SUBAPPLICATION Uebung_HystereseVertikal_AX_withAnalog (* MID/DEAD/HYSTERESIS-Eingabefelder bewegen live die 5 Schwellwert-Dreiecke im vertikalen Bargraph (Type=1 BottomToTop, Pixelposition gespiegelt: hoher Wert = kleiner Top) *)
  (* Standard: 61499-2; Description: Copyright (c) 2026 Meisterschulen am Ostbahnhof This program and the accompanying materials are made available under the terms of the Eclipse Public License 2.0 which is available at https://www.eclipse.org/legal/epl-2.0/ SPDX-License-Identifier: EPL-2.0 *)
  (* Version 1.1, 2026-09-27, Franz Höpfinger, Meisterschulen am Ostbahnhof, AR_TO_AI, Zero, QPos zu MyLib::sys::Q_ChildPosition_AR_Vertikal SubApp ausgelagert *)
  PACKAGE Uebungen;
  IMPORT Uebungen::const::UT::HystereseVertikal::DefaultPool_Numeric::InputNumber_MID_N;
  IMPORT Uebungen::const::UT::HystereseVertikal::DefaultPool_Numeric::InputNumber_DEAD_N;
  IMPORT Uebungen::const::UT::HystereseVertikal::DefaultPool_Numeric::InputNumber_HYSTERESIS_N;
  IMPORT Uebungen::const::UT::HystereseVertikal::DefaultPool::Polygon_MID;
  IMPORT Uebungen::const::UT::HystereseVertikal::DefaultPool::Polygon_MID_PLUS_DEAD;
  IMPORT Uebungen::const::UT::HystereseVertikal::DefaultPool::Polygon_MID_MINUS_DEAD;
  IMPORT Uebungen::const::UT::HystereseVertikal::DefaultPool::Polygon_MID_PLUS_DEAD_HYST;
  IMPORT Uebungen::const::UT::HystereseVertikal::DefaultPool::Polygon_MID_MINUS_DEAD_HYST;
  IMPORT Uebungen::const::UT::HystereseVertikal::DefaultPool::Container_Schwellwerte;
  IMPORT Uebungen::const::UT::HystereseVertikal::DefaultPool::NumberVariable_Istwert;
  IMPORT Uebungen::const::UT::HystereseVertikal::DefaultPool_Bargraph::Bargraph_Hysterese_ScalePx;
  IMPORT Uebungen::const::UT::HystereseVertikal::DefaultPool_Bargraph::Bargraph_Hysterese_LengthPx;
  IMPORT logiBUS::io::AI::logiBUS_AI::AnalogInput_I4;
  IMPORT logiBUS::io::DQ::logiBUS_DO::Output_Q1;
  IMPORT logiBUS::io::DQ::logiBUS_DO::Output_Q2;
  FBS
    MID_N : isobus::UT::io::NumericValue::NumericValue_PHYSA(QI := TRUE, stObj := InputNumber_MID_N);
    DEAD_N : isobus::UT::io::NumericValue::NumericValue_PHYSA(QI := TRUE, stObj := InputNumber_DEAD_N);
    HYST_N : isobus::UT::io::NumericValue::NumericValue_PHYSA(QI := TRUE, stObj := InputNumber_HYSTERESIS_N);
    Split_MID : adapter::events::unidirectional::AR_SPLIT_4;
    Split_DEAD : adapter::events::unidirectional::AR_SPLIT_3;
    Split_HYST : adapter::events::unidirectional::AR_SPLIT_3;
    Add_MidDead : adapter::iec61131::arithmetic::AR_ADD_2;
    Sub_MidDead : adapter::iec61131::arithmetic::AR_SUB_2;
    Split_AddResult : adapter::events::unidirectional::AR_SPLIT_2;
    Split_SubResult : adapter::events::unidirectional::AR_SPLIT_2;
    Add_MidDeadHyst : adapter::iec61131::arithmetic::AR_ADD_2;
    Sub_MidDeadHyst : adapter::iec61131::arithmetic::AR_SUB_2;
    AnalogInput_I4 : logiBUS::io::AI::logiBUS_AI_IDA(QI := TRUE, Input := AnalogInput_I4, AnalogInput_hysteresis := DWORD#0, TimeDelta := DWORD#250, TimeRateLimit := DWORD#100);
    AD_TO_AUDI : adapter::conversion::unidirectional::AD_TO_AUDI;
    AUDI_TO_AR : adapter::conversion::unidirectional::AUDI_TO_AR;
    Split_Istwert : adapter::events::unidirectional::AR_SPLIT_2;
    Q_Istwert : isobus::UT::Q::Q_NumericValue_PHYSA(stObj := (u16ObjId := NumberVariable_Istwert, r32Scale := 1.0, i32Offset := 0, u8Decimals := 0));
    DualHysteresis : logiBUS::signalprocessing::hysteresis::DualHysteresis_AR_AX(QI := TRUE);
    Output_Hoch : logiBUS::io::DQ::logiBUS_QXA(QI := TRUE, Output := Output_Q1);
    Output_Runter : logiBUS::io::DQ::logiBUS_QXA(QI := TRUE, Output := Output_Q2);
    BgLen_MID : adapter::types::unidirectional::AR::initval::initval_AR(INIT_VAL := Bargraph_Hysterese_LengthPx);
    SubFlip_MID : adapter::iec61131::arithmetic::AR_SUB_2;
    BgLen_MID_PLUS_DEAD : adapter::types::unidirectional::AR::initval::initval_AR(INIT_VAL := Bargraph_Hysterese_LengthPx);
    SubFlip_MID_PLUS_DEAD : adapter::iec61131::arithmetic::AR_SUB_2;
    BgLen_MID_MINUS_DEAD : adapter::types::unidirectional::AR::initval::initval_AR(INIT_VAL := Bargraph_Hysterese_LengthPx);
    SubFlip_MID_MINUS_DEAD : adapter::iec61131::arithmetic::AR_SUB_2;
    BgLen_MID_PLUS_DEAD_HYST : adapter::types::unidirectional::AR::initval::initval_AR(INIT_VAL := Bargraph_Hysterese_LengthPx);
    SubFlip_MID_PLUS_DEAD_HYST : adapter::iec61131::arithmetic::AR_SUB_2;
    BgLen_MID_MINUS_DEAD_HYST : adapter::types::unidirectional::AR::initval::initval_AR(INIT_VAL := Bargraph_Hysterese_LengthPx);
    SubFlip_MID_MINUS_DEAD_HYST : adapter::iec61131::arithmetic::AR_SUB_2;
  END_FBS
  SUBAPPS
    Mul_Istwert : MyLib::sys::AR_R_MUL(FACTOR := REAL#0.024420024420024420);
    Mul_MID : MyLib::sys::AR_R_MUL(FACTOR := Bargraph_Hysterese_ScalePx);
    QPos_MID : MyLib::sys::Q_ChildPosition_AR_Vertikal(u16ObjId := Polygon_MID, u16ObjIdParent := Container_Schwellwerte, xScale := TRUE);
    Mul_MID_PLUS_DEAD : MyLib::sys::AR_R_MUL(FACTOR := Bargraph_Hysterese_ScalePx);
    QPos_MID_PLUS_DEAD : MyLib::sys::Q_ChildPosition_AR_Vertikal(u16ObjId := Polygon_MID_PLUS_DEAD, u16ObjIdParent := Container_Schwellwerte, xScale := TRUE);
    Mul_MID_MINUS_DEAD : MyLib::sys::AR_R_MUL(FACTOR := Bargraph_Hysterese_ScalePx);
    QPos_MID_MINUS_DEAD : MyLib::sys::Q_ChildPosition_AR_Vertikal(u16ObjId := Polygon_MID_MINUS_DEAD, u16ObjIdParent := Container_Schwellwerte, xScale := TRUE);
    Mul_MID_PLUS_DEAD_HYST : MyLib::sys::AR_R_MUL(FACTOR := Bargraph_Hysterese_ScalePx);
    QPos_MID_PLUS_DEAD_HYST : MyLib::sys::Q_ChildPosition_AR_Vertikal(u16ObjId := Polygon_MID_PLUS_DEAD_HYST, u16ObjIdParent := Container_Schwellwerte, xScale := TRUE);
    Mul_MID_MINUS_DEAD_HYST : MyLib::sys::AR_R_MUL(FACTOR := Bargraph_Hysterese_ScalePx);
    QPos_MID_MINUS_DEAD_HYST : MyLib::sys::Q_ChildPosition_AR_Vertikal(u16ObjId := Polygon_MID_MINUS_DEAD_HYST, u16ObjIdParent := Container_Schwellwerte, xScale := TRUE);
  END_SUBAPPS
  ADAPTER_CONNECTIONS
    MID_N.rPhys TO Split_MID.IN;
    DEAD_N.rPhys TO Split_DEAD.IN;
    HYST_N.rPhys TO Split_HYST.IN;
    Split_MID.OUT2 TO Add_MidDead.IN1;
    Split_DEAD.OUT1 TO Add_MidDead.IN2;
    Split_MID.OUT3 TO Sub_MidDead.IN1;
    Split_DEAD.OUT2 TO Sub_MidDead.IN2;
    Add_MidDead.OUT TO Split_AddResult.IN;
    Sub_MidDead.OUT TO Split_SubResult.IN;
    Split_AddResult.OUT2 TO Add_MidDeadHyst.IN1;
    Split_HYST.OUT1 TO Add_MidDeadHyst.IN2;
    Split_SubResult.OUT2 TO Sub_MidDeadHyst.IN1;
    Split_HYST.OUT2 TO Sub_MidDeadHyst.IN2;
    AnalogInput_I4.IN TO AD_TO_AUDI.AD_IN;
    AD_TO_AUDI.AUDI_OUT TO AUDI_TO_AR.AUDI_IN;
    AUDI_TO_AR.AR_OUT TO Mul_Istwert.IN1;
    Mul_Istwert.OUT TO Split_Istwert.IN;
    Split_Istwert.OUT1 TO Q_Istwert.rPhys;
    Split_Istwert.OUT2 TO DualHysteresis.INPUT;
    Split_MID.OUT4 TO DualHysteresis.MI;
    Split_DEAD.OUT3 TO DualHysteresis.DEAD;
    Split_HYST.OUT3 TO DualHysteresis.HYSTERESIS;
    DualHysteresis.DO_UP TO Output_Hoch.OUT;
    DualHysteresis.DO_DOWN TO Output_Runter.OUT;
    Split_MID.OUT1 TO Mul_MID.IN1;
    BgLen_MID.OUT TO SubFlip_MID.IN1;
    Mul_MID.OUT TO SubFlip_MID.IN2;
    SubFlip_MID.OUT TO QPos_MID.rPhys;
    Split_AddResult.OUT1 TO Mul_MID_PLUS_DEAD.IN1;
    BgLen_MID_PLUS_DEAD.OUT TO SubFlip_MID_PLUS_DEAD.IN1;
    Mul_MID_PLUS_DEAD.OUT TO SubFlip_MID_PLUS_DEAD.IN2;
    SubFlip_MID_PLUS_DEAD.OUT TO QPos_MID_PLUS_DEAD.rPhys;
    Split_SubResult.OUT1 TO Mul_MID_MINUS_DEAD.IN1;
    BgLen_MID_MINUS_DEAD.OUT TO SubFlip_MID_MINUS_DEAD.IN1;
    Mul_MID_MINUS_DEAD.OUT TO SubFlip_MID_MINUS_DEAD.IN2;
    SubFlip_MID_MINUS_DEAD.OUT TO QPos_MID_MINUS_DEAD.rPhys;
    Add_MidDeadHyst.OUT TO Mul_MID_PLUS_DEAD_HYST.IN1;
    BgLen_MID_PLUS_DEAD_HYST.OUT TO SubFlip_MID_PLUS_DEAD_HYST.IN1;
    Mul_MID_PLUS_DEAD_HYST.OUT TO SubFlip_MID_PLUS_DEAD_HYST.IN2;
    SubFlip_MID_PLUS_DEAD_HYST.OUT TO QPos_MID_PLUS_DEAD_HYST.rPhys;
    Sub_MidDeadHyst.OUT TO Mul_MID_MINUS_DEAD_HYST.IN1;
    BgLen_MID_MINUS_DEAD_HYST.OUT TO SubFlip_MID_MINUS_DEAD_HYST.IN1;
    Mul_MID_MINUS_DEAD_HYST.OUT TO SubFlip_MID_MINUS_DEAD_HYST.IN2;
    SubFlip_MID_MINUS_DEAD_HYST.OUT TO QPos_MID_MINUS_DEAD_HYST.rPhys;
  END_CONNECTIONS
END_SUBAPPLICATION
